FUNCTION_BLOCK fbManipulatorContext EXTENDS TcoCore.TcoContext
VAR
    _automat : fbManipulatorAutomat(THIS^, eRestoreMode.AutoRestoreMembers);
END_VAR

METHOD PROTECTED Main
_automat();
END_METHOD

END_FUNCTION_BLOCK

(* stored: Version 1.1.0.1
   POU fbManipulatorContext: Id {ea90540b-6619-0c29-21fd-12c4e49ac96f}, SpecialFunc None
   Method Main: Id {cbd32a64-6d8a-060a-13a2-f1236a7a469f} *)
